{attribute 'qualified_only'}
{attribute 'strict'}
{attribute 'conditionalshow'}
TYPE E_ProfidriveGSM_State :
(
	S0_Disabled := 0,
	S1_SwitchingOnInhibited := 1,
	S2_ReadyForSwitchingOn := 2,
	S3_SwitchedOn := 3,
	S4_Operation := 4,
	S51_RampStop := 51,
	S52_QuickStop := 52
);
END_TYPE

(* stored: Version 1.1.0.1, ProductVersion 3.1.4024.12
   EnumerationTextList E_ProfidriveGSM_State: Id {59834f51-4abb-0c4d-159a-0c6125a4fbe5} *)
